Fanuc KAREL source: kc00009.KL

-- PROVISIONAL review KL for V940-1; original PC SHA256 8f98d48b63965e4d5cf437d5ffa3115c4b68d3e93f64405af45ec877f1f292a1
-- Incomplete behavior may be omitted. Consult companion uncertainty JSON. Do not deploy.
PROGRAM KC00009
%NOLOCKGROUP
BEGIN
  -- V9_ZERO_TABLE_METADATA_HINT layout=0002_ascii; no indexed target words; source/name/runtime held
  -- UNRESOLVED_PC offsets 5-33; opcodes 27,22,1C,22,22,31
  -- UNRESOLVED_PC offsets 38-42; opcodes 7F
END KC00009
